// TIA Portal V19 export
VAR_GLOBAL   // PLC tag table "HU_Area01_IO"
   HU_Area01_Pump_C AT %Q1.1 : Bool;   // 770KA1
   HU_Area01_Pump_Fdbk AT %I3.4 : Bool;   // 770KM1
   HU_Area01_S_LowLevel AT %I127.0 : Bool;   // 773SL1
   HU_Area01_S_LowLowLevel AT %I127.1 : Bool;   // 773SL2
   HU_Area01_S_ThermostatMax AT %I127.2 : Bool;   // 773SL3
   HU_Area01_S_ReturnFilterClogged AT %I127.3 : Bool;   // 773SL4
   HU_Area01_AI_Temperature AT %IW908 : Int;   // 464A1 - 773B1
   HU_Area01_AI_Pressure_CoilCar AT %IW910 : Int;   // 464A1 - 774B1
   HU_Area01_AI_Pressure_Peeler AT %IW912 : Int;   // 464A1 - 774B2
   HU_Area01_AI_Pressure_JB_Cut AT %IW914 : Int;   // 464A1 - 774B3
   HU_Area01_HeatExch_C AT %Q1.2 : Bool;   // 775QF1
   HU_Area01_HeatExch_Fdbk AT %I3.5 : Bool;   // 775KM1
END_VAR
